// TIA Portal V17 export
// export: Created 2022-07-20T07:01:30.5762896Z, ExportSetting WithDefaults, DisplayName Totally Integrated Automation Portal, DisplayVersion V17, DisplayName TIA Portal Openness, DisplayVersion V17, DisplayName TIA Portal Version Control Interface, DisplayVersion V17, DisplayName SINAMICS Startdrive Advanced, DisplayVersion V17, DisplayName SINAMICS Startdrive G130, G150, S120, S150, SINAMICS MV, S210, DisplayVersion V17, DisplayName SINAMICS Startdrive G110M, G120, G120C, G120D, G120P, G115D, DisplayVersion V17, DisplayName STEP 7 Professional, DisplayVersion V17, DisplayName STEP 7 Safety, DisplayVersion V17, DisplayName WinCC Advanced, DisplayVersion V17
FUNCTION_BLOCK "FB10040_Button_DetectPushType"   // FB10040, LAD
{ S7_Optimized_Access := 'TRUE' }
VERSION : 0.1
// stored: AutoNumber false, IsIECCheckEnabled false, IsRetainMemResEnabled false, MemoryReserve 100, SetENOAutomatically false, UDAEnableTagReadback false
   VAR_INPUT
      PushButton : Bool;
      MaxTimeShortPress : Time := T#1s;
   END_VAR
   VAR_OUTPUT
      ShortPressDetected : Bool;
      LongPressDetected : Bool;
      OnLongPress : Bool;
   END_VAR
   VAR
      TON_PushButton { S7_SetPoint := 'True'} : TON_TIME;
      TOF_PushButton { S7_SetPoint := 'True'} : TOF_TIME;
      TP_LongPress { S7_SetPoint := 'True'} : TP_TIME;
      TP_ShortPress { S7_SetPoint := 'True'} : TP_TIME;
      Rising_PushButton { ExternalAccessible := 'False'; ExternalVisible := 'False'; ExternalWritable := 'False'} : Bool;
   END_VAR
   VAR_TEMP   // added for the SCL form of the ladder/FBD networks
      _w1 : Bool;
   END_VAR
BEGIN

REGION Network 1: Long Press Detected
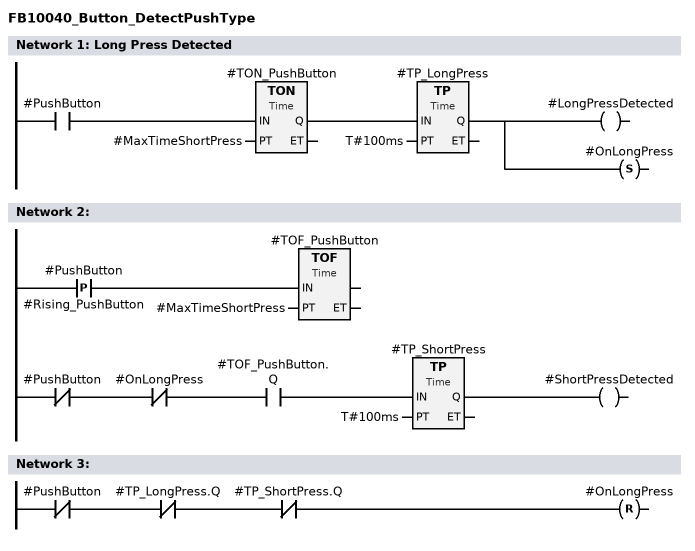
   RUNG wire#powerrail
      Contact( #PushButton )
      { S7_Templates := "time_type := Time" } #TON_PushButton.TON(pt := #MaxTimeShortPress, et =>)
      { S7_Templates := "time_type := Time" } #TP_LongPress.TP(pt := T#100ms, et =>)
      wire#w1
      Coil( #LongPressDetected )
   END_RUNG
   RUNG wire#w1
      S_Coil( #OnLongPress )
   END_RUNG
   // the same network as SCL:
   #TON_PushButton(IN := #PushButton, PT := #MaxTimeShortPress);   // TON
   #TP_LongPress(IN := #TON_PushButton.Q, PT := T#100ms);   // TP
   #LongPressDetected := #TP_LongPress.Q;
   IF #TP_LongPress.Q THEN #OnLongPress := TRUE; END_IF;
END_REGION

REGION Network 2
   RUNG wire#powerrail
      P_Contact(operand := #PushButton, bit := #Rising_PushButton)
      { S7_Templates := "time_type := Time" } #TOF_PushButton.TOF(pt := #MaxTimeShortPress, et =>)
   END_RUNG
   RUNG wire#powerrail
      I_Contact( #PushButton )
      I_Contact( #OnLongPress )
      Contact( #TOF_PushButton.Q )
      { S7_Templates := "time_type := Time" } #TP_ShortPress.TP(pt := T#100ms, et =>)
      Coil( #ShortPressDetected )
   END_RUNG
   // the same network as SCL:
   #_w1 := #PushButton AND NOT #Rising_PushButton;   // rising edge of #PushButton
   #Rising_PushButton := #PushButton;
   #TOF_PushButton(IN := #_w1, PT := #MaxTimeShortPress);   // TOF
   #TP_ShortPress(IN := NOT #PushButton AND NOT #OnLongPress AND #TOF_PushButton.Q, PT := T#100ms);   // TP
   #ShortPressDetected := #TP_ShortPress.Q;
END_REGION

REGION Network 3
   RUNG wire#powerrail
      I_Contact( #PushButton )
      I_Contact( #TP_LongPress.Q )
      I_Contact( #TP_ShortPress.Q )
      R_Coil( #OnLongPress )
   END_RUNG
   // the same network as SCL:
   IF NOT #PushButton AND NOT #TP_LongPress.Q AND NOT #TP_ShortPress.Q THEN #OnLongPress := FALSE; END_IF;
END_REGION
END_FUNCTION_BLOCK
